// TIA Portal V18 export
TYPE "PLCtoMES_OP_ProcessData_OP220"
// stored: IsFailsafeCompliant false
   STRUCT
      DATA : Real;
   END_STRUCT;
END_TYPE
